ABB RobotStudio station: Celda_Robotizada_Soldadura.rsstn

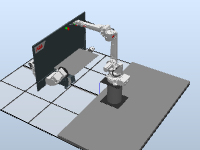
Station Celda_Robotizada_Soldadura (saved by RobotStudio 20.4.9280.0)
Controller Controlador, task T_ROB1: task frame (RAPID world) sits at (500, 0, 800) mm, rotated rx 0 ry 0 rz 180 deg in the station
Controller Controlador
  mechanical unit INTERCH: IRBP_R300_D1000-L1250_M2009_REV1_01, 3 joints, base frame (0, 0, 0) mm
  mechanical unit STN1: IRBP_R300_D1000-L1250_M2009_REV1_01, 1 joints, base frame (1710, -600, 150) mm, rotated rx 0 ry -90 rz -90 deg
  mechanical unit STN2: IRBP_R300_D1000-L1250_M2009_REV1_01, 1 joints, base frame (0, 0, 0) mm
  mechanical unit ROB_1: IRB2600ID_8_200__03, 6 joints, base frame (0, 0, 0) mm
Layout (positions relative to the parent item):
  - Pieza_1 [part]
  - IRBP_R300_D1000-L1250_M2009_REV1_01 [mechanism] at (-1800, 625, 0) mm; joint values [0, 0, 0] (rad or m)
      links: Base, Link1, Link2, Link3
  - IRB2600ID_8_200__03 [mechanism, from Robots\IRB2600ID_8_200_G_03.rslib] at (500, 0, 800) mm, rotated rx 0 ry 0 rz 180 deg; joint values [0, 0, 0, 0, 0.5236, 0] (rad or m)
  - Pieza_2 [part] at (0, 0, 100) mm
  - Pieza_4 [part] at (0, 0, 100) mm
  - Pieza_6 [part] at (0, 0, 793) mm
  - Binzel_ID_22 [mechanism, from Tools\Binzel_ID_22.rslib] at (-761.21, 0, 2195) mm, rotated rx 180 ry 60 rz 0 deg
  - Pieza_7 [part] at (70, 0, 950) mm
Attachment: Binzel_ID_22 is attached to IRB2600ID_8_200__03 / Link6
Targets, tools, work objects and paths stored in the station, written as RAPID:
! task T_ROB1
MODULE CalibData
  PERS tooldata tWeldGun:=[TRUE,[[49.841566361,0,372.194826196],[0.981627183,0,0.190808995,0]],[2,[0,0,100],[0,1,0,0],0,0,0]];
ENDMODULE

